Staubli VAL3: onF7Event.pgx

program onF7Event()
begin
   // look if the bButton is enable
  if bButton[6]
    //
  endIf
   end
